// SIMATIC S7-200 project (STEP 7-Micro/WIN), CPU 224XP CN REL 02.01

ORGANIZATION_BLOCK MAIN:OB1
TITLE=PROGRAM COMMENTS
BEGIN
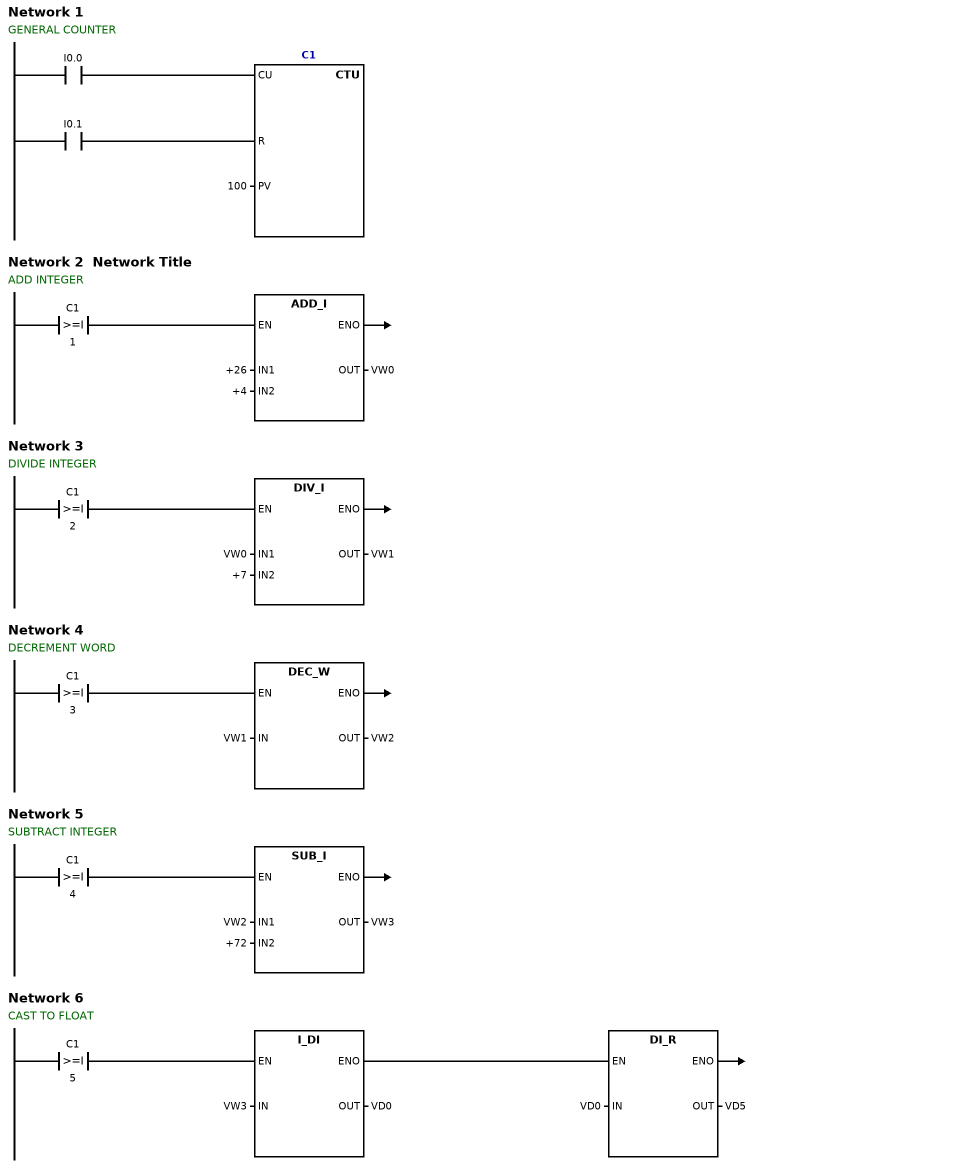
Network 1
// GENERAL COUNTER
LD     I0.0
LD     I0.1
CTU    C1, 100
Network 2 // Network Title
// ADD INTEGER
LDW>=  C1, 1
MOVW   +26, VW0
+I     +4, VW0
Network 3
// DIVIDE INTEGER
LDW>=  C1, 2
MOVW   VW0, VW1
/I     +7, VW1
Network 4
// DECREMENT WORD
LDW>=  C1, 3
MOVW   VW1, VW2
DECW   VW2
Network 5
// SUBTRACT INTEGER
LDW>=  C1, 4
MOVW   VW2, VW3
-I     +72, VW3
Network 6
// CAST TO FLOAT
LDW>=  C1, 5
ITD    VW3, VD0
AENO
DTR    VD0, VD5
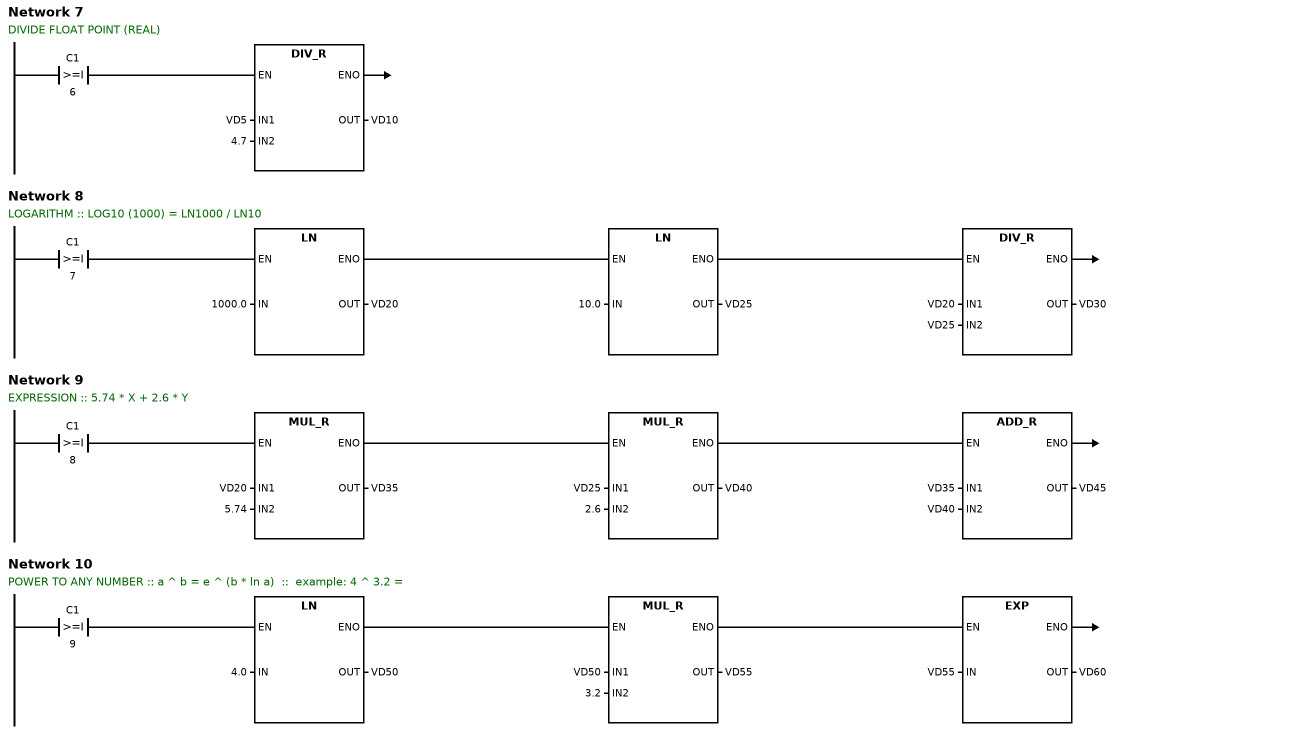
Network 7
// DIVIDE FLOAT POINT (REAL)
LDW>=  C1, 6
MOVR   VD5, VD10
/R     4.7, VD10
Network 8
// LOGARITHM :: LOG10 (1000) = LN1000 / LN10
LDW>=  C1, 7
LN     1000.0, VD20
AENO
LN     10.0, VD25
AENO
MOVR   VD20, VD30
/R     VD25, VD30
Network 9
// EXPRESSION :: 5.74 * X + 2.6 * Y
LDW>=  C1, 8
MOVR   VD20, VD35
AENO
*R     5.74, VD35
AENO
MOVR   VD25, VD40
AENO
*R     2.6, VD40
AENO
MOVR   VD35, VD45
+R     VD40, VD45
Network 10
// POWER TO ANY NUMBER :: a ^ b = e ^ (b * ln a)  ::  example: 4 ^ 3.2 = 
LDW>=  C1, 9
LN     4.0, VD50
AENO
MOVR   VD50, VD55
AENO
*R     3.2, VD55
AENO
EXP    VD55, VD60
END_ORGANIZATION_BLOCK
